(*

.. <legal notes>

legal notes
=================
| SPDX-FileCopyrightText: © 2025 Oleksandr Tiutyk <trofimich@gmail.com>
| SPDX-License-Identifier: LGPL-3.0-only
| For details check: LGPL-3.0-only_

.. _LGPL-3.0-only: https://www.gnu.org/licenses/lgpl-3.0.en.html

.. </legal notes>

*)

{attribute 'no_explicit_call' := 'do not call this function block directly'} 
FUNCTION_BLOCK ABSTRACT Process EXTENDS Object IMPLEMENTS IProcess
VAR
	_StateChanged : BOOL;
	
	_Running : BOOL;
	
	_Error : BOOL;	
	_ErrorMessage : ERROR_MESSAGE;
END_VAR

{attribute 'monitoring' := 'call'}
{attribute 'OPC.UA.DA.Property' := '1'}
{attribute 'OPC.UA.DA.Access' := '1'}
PROPERTY FINAL Error : BOOL
GET
Error := _Error;
END_GET
END_PROPERTY

{attribute 'monitoring' := 'call'}
{attribute 'OPC.UA.DA.Property' := '1'}
{attribute 'OPC.UA.DA.Access' := '1'}
PROPERTY FINAL ErrorMessage : REFERENCE TO ERROR_MESSAGE
GET
ErrorMessage REF= _ErrorMessage;
END_GET
END_PROPERTY

METHOD FINAL Execute 
VAR
	exceptionCode : __SYSTEM.ExceptionCode;
END_VAR
_StateChanged := FALSE;

__TRY
	IF Running THEN
		OnRunning(FALSE);
	END_IF
__CATCH(exceptionCode)
	handleException(exceptionCode);
__ENDTRY
END_METHOD

METHOD PRIVATE handleException
VAR_INPUT
	exceptionCode : __SYSTEM.ExceptionCode;
END_VAR
VAR
	exception : IException;
END_VAR
exception := ExceptionManager.GetLastException(exceptionCode);

__TRY
	OnError();
__CATCH
__ENDTRY

_ErrorMessage := exception.GetMessage();
	
IF NOT _Error THEN
	LogManager.TryLogMessage(WideStringHelper.ConcatStrings255("Process '", Name, "' failed at ", TO_WSTRING(SystemDateTimeManager.SystemLocalDateTime)), LOG_CATEGORY.SUCCESS, TO_WSTRING(ClassName), "Process", "ProcessFailed");
	
	_StateChanged := TRUE;
END_IF

_Running := FALSE;
_Error := TRUE;

ExceptionManager.Throw(exception);
END_METHOD

{attribute 'monitoring' := 'call'}
{attribute 'OPC.UA.DA.Property' := '1'}
{attribute 'OPC.UA.DA.Access' := '1'}
PROPERTY ABSTRACT Name : WSTRING
GET
END_GET
END_PROPERTY

METHOD PROTECTED OnError
END_METHOD

METHOD PROTECTED ABSTRACT OnRunning 
VAR_INPUT
	isStart : BOOL;
END_VAR
END_METHOD

{attribute 'monitoring' := 'call'}
{attribute 'OPC.UA.DA.Property' := '1'}
{attribute 'OPC.UA.DA.Access' := '1'}
PROPERTY FINAL Running : BOOL
GET
Running := _Running;
END_GET
END_PROPERTY

METHOD PRIVATE FINAL setRunningState
IF NOT _Running THEN
	LogManager.TryLogMessage(WideStringHelper.ConcatStrings255("Process '", Name, "' started at ", TO_WSTRING(SystemDateTimeManager.SystemLocalDateTime)), LOG_CATEGORY.SUCCESS, TO_WSTRING(ClassName), "Process", "ProcessStarted");
	
	_StateChanged := TRUE;
END_IF

_Running := TRUE;

_Error := FALSE;
_ErrorMessage := "";
END_METHOD

METHOD FINAL Start
VAR
	exceptionCode : __SYSTEM.ExceptionCode;
	
	exception : IException;

	errorMessage : ERROR_MESSAGE;	
END_VAR
__TRY
	setRunningState();
				
	OnRunning(TRUE);
__CATCH(exceptionCode)
	handleException(exceptionCode);
__ENDTRY
END_METHOD

{attribute 'monitoring' := 'call'}
{attribute 'OPC.UA.DA.Property' := '1'}
{attribute 'OPC.UA.DA.Access' := '1'}
PROPERTY FINAL StateChanged : BOOL
GET
StateChanged := _StateChanged;
END_GET
END_PROPERTY

END_FUNCTION_BLOCK

(* stored: Version 1.1.0.1
   POU Process: Id {cf0466a4-6c52-4c7f-8d30-0762e3c9f951}, SpecialFunc None
   Folder Members to override: Id {f0437e52-a6e0-457b-b826-a1b0d3aa42e4}
   Folder Service members: Id {f24b970a-f6c5-4810-b7f1-6c973b901a78}
   Property Error: Id {cba50b93-ca87-4893-b8e0-4db492fd2b93}
   Get Get: Id {c33c83f5-a7b9-43fc-80ed-8782730cbd21}
   Property ErrorMessage: Id {5f4f1fa0-e186-4cdb-b4b0-72e44dd875e0}
   Get Get: Id {53d45b00-4d01-4a78-a143-e8855149b365}
   Method Execute: Id {8cb4c5e0-e266-49dd-8b13-3992f844cd79}
   Method handleException: Id {67e1128a-d723-47b1-a342-34f878a20566}
   Property Name: Id {5b4d37f8-0df9-4be8-9516-8aee2f6e0819}
   Get Get: Id {49c90946-6b6a-4a0c-af79-95ca349a4b22}
   Method OnError: Id {ee41bc9e-7ec2-4e2c-8ebf-acedded1d8f4}
   Method OnRunning: Id {4c9b8028-0b09-4527-b769-cd260bab25d2}
   Property Running: Id {646acde6-23db-47a0-a4a5-3d9ed68337d1}
   Get Get: Id {85a56550-0022-468b-93e5-b71c92daf8d4}
   Method setRunningState: Id {9d107778-1f40-457f-bb67-dcb48cbf13a9}
   Method Start: Id {ffda977e-9b04-49e3-ae34-eee8276e4ca5}
   Property StateChanged: Id {62596c98-537e-4a13-9120-67a983719c3b}
   Get Get: Id {26160b98-5b31-490e-b967-87ec988d603a} *)
